// TIA Portal V19 export
TYPE "LAF_typeJobsInterface"
TITLE = LAF_typeJobInterface
// Interface to control jobs from an HMI
// stored: Access Published
   STRUCT
      commands { S7_SetPoint := 'True'} : "LAF_typeJobsCommands";
      status { S7_SetPoint := 'True'} : "LAF_typeJobsStatus";   // Control of the Job Management
   END_STRUCT;
END_TYPE
